# B&R Automation Studio project PloterCNC
Automation Studio 4.7.3.93 SP; technology packages: mapp 5.10.1, mappCockpit 5.10.1, mappControl 5.10.0, mappMotion 5.10.1, mappView 5.10.1

## Configuration PloterCNC

CPU X20CP3584, AutomationRuntime C4.72, Build 4.1.2, Safety 0.0, Vc V4.72.0

### Task classes (Cpu.sw)
```
Cyclic#2:
  Program <- Program.prg
DataObjects: McAcpSys
NcDataObjects: CncProg <- CncProg.dob, CncSquare <- CncSquare.dob
Binaries: udbdef, arsvcreg, FWRules, McAcpDrv, McMechSys, McAcpSim, mvLoader, mCoWebSc, TCData, arflatprv, arcoal, iomap, Config_4, asfw, Config_3, Role, Config_1, Config_2, arconfig, ashwd, Hierarchy, sysconf, User, ashwac
Libraries: McBase, MpCnc, MpBase, McAxGroup, McPathGen, McAxis, McProgInt, McAcpAx, CoTrace, AsZip, FileIO, runtime, asmem, sys_lib, arssl, asarprof, powerlnk, asieccon, dataobj, brsystem, asarlog, MpAlarmX, astime, MpServer
```

### Hardware
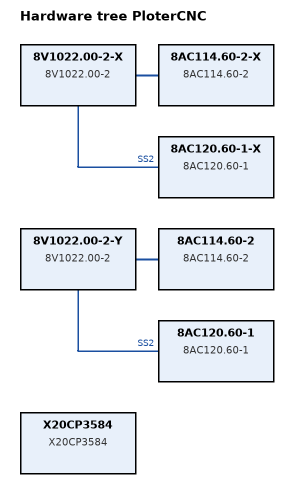
```
8AC114.60-2 : 8AC114.60-2 v1.0.0.8  [SS -> 8V1022.00-2-Y.SS1; PLK1 -> 8AC114.60-2-X.PLK2 [Cable Type=PowerlinkCable, Length=10, Version=1.0.0.2]]
8AC114.60-2-X : 8AC114.60-2 v1.0.0.8  [SS -> 8V1022.00-2-X.SS1; PLK1 -> X20CP3584.IF3 [Cable Type=PowerlinkCable, Length=10, Version=1.0.0.2]; PLK2 -> 8AC114.60-2.PLK1 [Cable Type=PowerlinkCable, Length=10, Version=1.0.0.2]]
8AC120.60-1 : 8AC120.60-1 v2.2.0.0  [SS -> 8V1022.00-2-Y.SS2]
  PlugInType = Encoder
  McAcoposTypeID = AcoposPlugInConfig
8AC120.60-1-X : 8AC120.60-1 v2.2.0.0  [SS -> 8V1022.00-2-X.SS2]
  PlugInType = Encoder
  McAcoposTypeID = AcoposPlugInConfig
8V1022.00-2-X : 8V1022.00-2 v2.2.0.0
  DriveConfiguration/Module:
    McAcoposTypeID = AcoposConfig
    ActivateACOPOSSimulationOnPLC = 0
  DriveConfiguration/Channel[1]/RealAxis:
    AxisReference = gAxisQX
  DriveConfiguration/Channel[1]/RealAxis/MechanicalElements/Gearbox:
    InputIsReadOnly = 0
    Input = 1
    OutputIsReadOnly = 0
    Output = 1
  DriveConfiguration/Channel[1]/RealAxis/MechanicalElements/RotaryToLinearTransformation:
    ReferenceDistanceIsReadOnly = 0
    ReferenceDistance = 1.385
  DriveConfiguration/Channel[1]/RealAxis/Controller:
    ModeIsReadOnly = 0
    Mode = PositionController
  DriveConfiguration/Channel[1]/RealAxis/Controller/Mode/Position:
    ProportionalGain = 454
    IntegrationTime = 0.0
    PredictionTime = 0.0004
    TotalDelayTime = 0.0004
  DriveConfiguration/Channel[1]/RealAxis/Controller/Mode/Speed:
    ProportionalGainIsReadOnly = 0
    ProportionalGain = 0.6499999
    IntegrationTimeIsReadOnly = 0
    IntegrationTime = 0.0
    FilterTimeIsReadOnly = 0
    FilterTime = 0.0
  DriveConfiguration/Channel[1]/RealAxis/Controller/Mode/LoopFilters:
    LoopFilter1 = NotUsed
    LoopFilter2 = NotUsed
    LoopFilter3 = NotUsed
  DriveConfiguration/Channel[1]/RealAxis/Homing:
    Mode = AbsoluteCorrection
  DriveConfiguration/Channel[1]/RealAxis/Homing/Mode:
    Position = -223
  DriveConfiguration/Channel[1]/RealAxis/Homing:
    RestorePositionVariable = 
  DriveConfiguration/Channel[1]/RealAxis/StopReaction:
    Quickstop = DecelerationLimit
    DriveError = DecelerationLimit
  DriveConfiguration/Channel[1]/RealAxis/MovementErrorLimits:
    PositionError = 1.0
    VelocityErrorMonitoring = Automatic1
  DriveConfiguration/Channel[1]/RealAxis:
    JerkFilter = NotUsed
  DriveConfiguration/Channel[1]/RealAxis/DigitalInputs/HomingSwitch:
    Level = High
  DriveConfiguration/Channel[1]/RealAxis/DigitalInputs/PositiveLimitSwitch:
    Level = Low
  DriveConfiguration/Channel[1]/RealAxis/DigitalInputs/NegativeLimitSwitch:
    Level = Low
  DriveConfiguration/Channel[1]/RealAxis/DigitalInputs/Trigger1:
    Level = High
  DriveConfiguration/Channel[1]/RealAxis/DigitalInputs/Trigger2:
    Level = High
  DriveConfiguration/Channel[1]/RealAxis/DigitalInputs/Quickstop:
    Input = Trigger2
  DriveConfiguration/Channel[1]/RealAxis/Simulation:
    SimulationModeOnPLC = SetValueGeneration
    SimulationModeOnACOPOS = NotUsed
8V1022.00-2-Y : 8V1022.00-2 v2.2.0.0
  DriveConfiguration/Module:
    McAcoposTypeID = AcoposConfig
    ActivateACOPOSSimulationOnPLC = 0
  DriveConfiguration/Channel[1]/RealAxis:
    AxisReference = gAxisQY
  DriveConfiguration/Channel[1]/RealAxis/MechanicalElements/Gearbox:
    InputIsReadOnly = 0
    Input = 1
    OutputIsReadOnly = 0
    Output = 1
  DriveConfiguration/Channel[1]/RealAxis/MechanicalElements/RotaryToLinearTransformation:
    ReferenceDistanceIsReadOnly = 0
    ReferenceDistance = 1.385
  DriveConfiguration/Channel[1]/RealAxis/Controller:
    ModeIsReadOnly = 0
    Mode = PositionController
  DriveConfiguration/Channel[1]/RealAxis/Controller/Mode/Position:
    ProportionalGain = 496
    IntegrationTime = 0.0
    PredictionTime = 0.0004
    TotalDelayTime = 0.0004
  DriveConfiguration/Channel[1]/RealAxis/Controller/Mode/Speed:
    ProportionalGainIsReadOnly = 0
    ProportionalGain = 0.8499999
    IntegrationTimeIsReadOnly = 0
    IntegrationTime = 0.0
    FilterTimeIsReadOnly = 0
    FilterTime = 0.0
  DriveConfiguration/Channel[1]/RealAxis/Controller/Mode/LoopFilters:
    LoopFilter1 = NotUsed
    LoopFilter2 = NotUsed
    LoopFilter3 = NotUsed
  DriveConfiguration/Channel[1]/RealAxis/Homing:
    Mode = AbsoluteCorrection
  DriveConfiguration/Channel[1]/RealAxis/Homing/Mode:
    Position = 1761
  DriveConfiguration/Channel[1]/RealAxis/Homing:
    RestorePositionVariable = 
  DriveConfiguration/Channel[1]/RealAxis/StopReaction:
    Quickstop = DecelerationLimit
    DriveError = DecelerationLimit
  DriveConfiguration/Channel[1]/RealAxis/MovementErrorLimits:
    PositionError = 1.0
    VelocityErrorMonitoring = Automatic1
  DriveConfiguration/Channel[1]/RealAxis:
    JerkFilter = NotUsed
  DriveConfiguration/Channel[1]/RealAxis/DigitalInputs/HomingSwitch:
    Level = High
  DriveConfiguration/Channel[1]/RealAxis/DigitalInputs/PositiveLimitSwitch:
    Level = Low
  DriveConfiguration/Channel[1]/RealAxis/DigitalInputs/NegativeLimitSwitch:
    Level = Low
  DriveConfiguration/Channel[1]/RealAxis/DigitalInputs/Trigger1:
    Level = High
  DriveConfiguration/Channel[1]/RealAxis/DigitalInputs/Trigger2:
    Level = High
  DriveConfiguration/Channel[1]/RealAxis/DigitalInputs/Quickstop:
    Input = Trigger2
  DriveConfiguration/Channel[1]/RealAxis/Simulation:
    SimulationModeOnPLC = SetValueGeneration
    SimulationModeOnACOPOS = NotUsed
X20CP3584 : X20CP3584 v1.6.0.0
  Connector IF2:
    ActivateDevice = 1
    Mode = Manual
    InternetAddress = 10.0.0.2
    SubnetMask = 255.255.255.0
  Connector IF3:
    Channel1
    ChannelID1 = McAcpBroadcast
    ChannelType1 = OCTET[96]
  ConfigurationID = PloterCNC_PloterCNC
  UserPartitionSize = 100
  Simulation = 1
  TimerDeviceType = EPLX2X
  TimerDevice = X20CP3584.IF3
  TaskClassIdleTime = 2000
  Cyclic1Duration = 2000
  Cyclic1Tolerance = 0
  FtpUser1
  FtpUsername1 = admin
  FtpUserPassword1 = uWZf7lfkDMUZL52pN0YGjFsSlLYs7TnNYj8rJpA5ubQ=  // admin
  FtpUserSalt1 = 89IIsKuO
  FTPAccessRight1 = 0
  ActivateOpcUa = 1
  OpcUaInformationModels_PV_Version = 1
```

### Config_1.axesgroup - X20CP3584/mappMotion/2AxesCNCXY/Config_1.axesgroup
```
Element gCncXY (Type=axesgroup)
  Type = PathGenAxesGroup
    ProcessingTaskClass = 1
    License = 1
    PhysicalAxes:
      JointAxes:
        JointAxis[1]:
          Name = QX
          AxisRef = gAxisQX
        JointAxis[2]:
          Name = QY
          AxisRef = gAxisQY
    MechanicalSystem:
      MechSysRef = MechSys_2AxCNCXY
    BasicSettings:
      ModalDataBehaviour = ResetToDefault
      GeometryPlanning:
        RoundingMode = Standard
        MaxCornerDeviation = 0.0
        MaxTangentialTransitionDeviation = 0.0
        MaxRadiusDeviation = 0.001
        WorkingPlane = XY
      TrajectoryPlanning = Basic
        LimitCheckResolution = UserDefinedTime
          Time = 0.01
        BufferTime = UserDefinedTime
          Time = 0.1
    AxesGroupFeatures:
      FeatureRef[1] = Feature_Programs
      FeatureRef[2] = Feature_Jogging
  Alarms = None
```

### Config_2.axis - X20CP3584/mappMotion/2AxesCNCXY/Config_2.axis
```
Element gAxisQX (Type=axis)
  BaseTypeIsReadOnly = 0
  BaseType = LinearBounded
    MeasurementUnit = 5066068
    MeasurementResolutionIsReadOnly = 0
    MeasurementResolution = 0.01
    CountDirectionIsReadOnly = 0
    CountDirection = Standard
  MovementLimitsIsReadOnly = 0
  MovementLimits = Internal
    Position:
      LowerLimitMin = -1.79769313486231E308
      UpperLimitMax = 1.79769313486231E308
      LowerLimit = -10
      UpperLimit = 540
    VelocityIsReadOnly = 0
    Velocity:
      VelocityMax = 3.4E38
      Velocity = 100
    AccelerationIsReadOnly = 0
    Acceleration:
      AccelerationMax = 3.4E38
      Acceleration = 1000
    DecelerationIsReadOnly = 0
    Deceleration:
      DecelerationMax = 3.4E38
      Deceleration = 1000
  Alarms = None
Element gAxisQY (Type=axis)
  BaseTypeIsReadOnly = 0
  BaseType = LinearBounded
    MeasurementUnit = 5066068
    MeasurementResolutionIsReadOnly = 0
    MeasurementResolution = 0.01
    CountDirectionIsReadOnly = 0
    CountDirection = Inverse
  MovementLimitsIsReadOnly = 0
  MovementLimits = Internal
    Position:
      LowerLimitMin = -1.79769313486231E308
      UpperLimitMax = 1.79769313486231E308
      LowerLimit = -10
      UpperLimit = 410
    VelocityIsReadOnly = 0
    Velocity:
      VelocityMax = 3.4E38
      Velocity = 100
    AccelerationIsReadOnly = 0
    Acceleration:
      AccelerationMax = 3.4E38
      Acceleration = 1000
    DecelerationIsReadOnly = 0
    Deceleration:
      DecelerationMax = 3.4E38
      Deceleration = 1000
  Alarms = None
```

### Config_3.mechanicalsystem - X20CP3584/mappMotion/2AxesCNCXY/Config_3.mechanicalsystem
```
Element MechSys_2AxCNCXY (Type=mechanicalsystem)
  Type = 2AxesCNC
    Subtype = 2AxesCNCXY
      CoordinatesNames = Default
        XCoordinateName = X
        YCoordinateName = Y
      WireFrameModel = Standard
        FlangeToTcp = ConnectionLine
          Distance = 0.0
      JointAxesPositionLimits:
        JointAxis[1] = UseAxisLimits
        JointAxis[2] = UseAxisLimits
```

### Config_4.axesgroupfeature - X20CP3584/mappMotion/2AxesCNCXY/Config_4.axesgroupfeature
```
Element Feature_Programs (Type=axesgroupfeature)
  Type = Program
    ModalDataBehaviour = UseAxesGroupSettings
    InitialSettings:
      InterpolationTypes = LinearRapid
      PositionCoordinates = Absolute
      CircleCoordinates = Relative
      JACS_ACSProgramming = JACS
      ContourConnection = Inactive
      ProgrammingUnits = UseAxesGroupSettings
      Feedrates:
        FeedCharacteristic = StandardCharacteristic
        FeedType = Feedrate
        FeedReduction = Inactive
        FeedrateValue = 0.0
        InverseFeedrateValue = 0.0
        FeedratePerRevValue = 0.0
    DefaultLanguage = BRGCode
    Location = Default
      FileDevice = CNC_PrgDir
Element Feature_Jogging (Type=axesgroupfeature)
  Type = Jogging
```

### Config.mpalarmxcore - X20CP3584/mappServices/Config.mpalarmxcore
```
Element gAlarmXCore (Type=mpalarmxcore)
  mapp.AlarmX.Core.Configuration:
    [0]:
      Name = XAxisOutOfBounds
      Message = X axis went out of bounds!
      Behavior = LevelMonitoring
        Monitoring:
          MonitoredPV = ::Program:MpCnc2Axis_0.X
          LowLimitEnable = Static
            Limit = 0
          HighLimitEnable = Static
            Limit = 540
    [1]:
      Name = UserAlarm
      Message = This alarm is set by user!
      Behavior = PersistentAlarm
```

## Logical view

Binary libraries used (declarations not repeated): operator, runtime, astime, AsIecCon, McBase, MpCnc 5.10.1, MpBase, McAxGroup 5.10.1, McPathGen 5.10.1, McAxis, McProgInt 5.10.1, McAcpAx, CoTrace, AsZip, FileIO, MpAlarmX 5.10.1, MpServer 5.10.0


### Data object Logical/CncProg (Cnc)

#### CncProg.cnc - CNC program (G-Code)
```
%001 (CncProgram)

N10 G90     (absolute coordinates)
N20 F3000    (Feed rate in measurements units/min)

N30 G04 2   (dwell time 2s)

N50 G01 X80 Y100  (linear move)

N60 G04 2         (dwell time 2s)

N100 G00 X0 Y0    (rapid move to zero)
N999 M30
```

### Program Logical/Program (IEC)

#### Types.typ
```iecst
TYPE
	MotionStep_type :
		(
		STEP_INIT,
		STEP_POWER,
		STEP_HOME,
		STEP_AWAIT,
		STEP_RUN_PROGRAM,
		STEP_PROGRAM_INTERRUPTED,
		STEP_MOVE_Y_AXIS,
		STEP_MOVE_X_AXIS,
		STEP_ERROR
		);
END_TYPE
```

#### Variables.var
```iecst
VAR
	MpAlarmXHistory_0 : MpAlarmXHistory;
	MpAlarmXCore_0 : MpAlarmXCore;
	MpCnc2Axis_0 : MpCnc2Axis;
	CncParameters : MpCnc2AxisParType;
	MotionStep : MotionStep_type;
	ProgramOption : BOOL;
	AxisVelocity : REAL := 0.0;
END_VAR
(*Comands*)
VAR
	diErrorReset : BOOL;
	diRunProgram : BOOL;
	diResumeProgram : BOOL;
	diInterruptProgram : BOOL;
	diIncreaseYAxis : BOOL;
	diDecreaseYAxis : BOOL;
	diIncreaseXAxis : BOOL;
	diDecreaseXAxis : BOOL;
	diStop : BOOL;
	diStart : BOOL;
END_VAR
```

#### Main.st
```iecst
PROGRAM _INIT
	MpAlarmXCore_0.MpLink := ADR(gAlarmXCore);
	MpAlarmXCore_0.Enable := TRUE;

	MpAlarmXHistory_0.MpLink := ADR(gAlarmXHistory);
	MpAlarmXHistory_0.Enable := TRUE;

	MpCnc2Axis_0.MpLink := ADR(gCncXY);
	MpCnc2Axis_0.Enable := TRUE;
	MpCnc2Axis_0.Parameters := ADR(CncParameters);

	MpCnc2Axis_0.Override := 100.0;
	AxisVelocity := 0;
	CncParameters.Jog.Velocity[0] := AxisVelocity;
	CncParameters.Jog.Velocity[1] := AxisVelocity;
END_PROGRAM

PROGRAM _CYCLIC

	IF ProgramOption THEN
		CncParameters.ProgramName := 'CncSquare';
	ELSE
		CncParameters.ProgramName := 'CncProg';
	END_IF;

	MpCnc2Axis_0.ErrorReset := diErrorReset;

	IF EDGEPOS(MpCnc2Axis_0.Error) THEN
		MotionStep := STEP_ERROR;
	END_IF;

	CASE MotionStep OF
		STEP_INIT:
			MpCnc2Axis_0.Power := FALSE;
			MpCnc2Axis_0.Home := FALSE;

			IF diStart THEN
				MotionStep := STEP_POWER;
			END_IF;
		STEP_POWER:
			MpCnc2Axis_0.Power := TRUE;

			IF MpCnc2Axis_0.PowerOn THEN
				MotionStep := STEP_HOME;
			END_IF;
		STEP_HOME:
			MpCnc2Axis_0.Home := TRUE;

			IF MpCnc2Axis_0.IsHomed THEN
				MotionStep := STEP_AWAIT;
			END_IF;
		STEP_AWAIT:

			IF diStop THEN
	  			MotionStep := STEP_INIT;
			ELSIF diRunProgram THEN
				MotionStep := STEP_RUN_PROGRAM;
			ELSIF diIncreaseXAxis THEN
				CncParameters.Jog.Velocity[0] := AxisVelocity;
				MotionStep := STEP_MOVE_X_AXIS;
			ELSIF diDecreaseXAxis THEN
				CncParameters.Jog.Velocity[0] := -AxisVelocity;
				MotionStep := STEP_MOVE_X_AXIS;
			ELSIF diIncreaseYAxis THEN
				CncParameters.Jog.Velocity[1] := AxisVelocity;
				MotionStep := STEP_MOVE_Y_AXIS;
			ELSIF diDecreaseYAxis THEN
				CncParameters.Jog.Velocity[1] := -AxisVelocity;
				MotionStep := STEP_MOVE_Y_AXIS;
			END_IF;
		STEP_RUN_PROGRAM:
			MpCnc2Axis_0.MoveProgram := TRUE;
			MpCnc2Axis_0.Continue := FALSE;

			IF MpCnc2Axis_0.MoveDone THEN
				MotionStep := STEP_AWAIT;
				MpCnc2Axis_0.MoveProgram := FALSE;
			END_IF;

			IF diInterruptProgram THEN
				MotionStep := STEP_PROGRAM_INTERRUPTED;
			END_IF;
		STEP_PROGRAM_INTERRUPTED:
			MpCnc2Axis_0.Interrupt := TRUE;

			IF diResumeProgram THEN
				MotionStep := STEP_RUN_PROGRAM;
				MpCnc2Axis_0.Interrupt := FALSE;
				MpCnc2Axis_0.Continue := TRUE;
			END_IF;
		STEP_MOVE_X_AXIS:
			MpCnc2Axis_0.Jog := TRUE;

			IF NOT(diIncreaseXAxis) AND NOT(diDecreaseXAxis) THEN
				MotionStep := STEP_AWAIT;
				MpCnc2Axis_0.Jog := FALSE;
				CncParameters.Jog.Velocity[0] := 0;
			END_IF;
		STEP_MOVE_Y_AXIS:
			MpCnc2Axis_0.Jog := TRUE;

			IF  NOT(diIncreaseYAxis) AND NOT(diDecreaseYAxis) THEN
				MotionStep := STEP_AWAIT;
				MpCnc2Axis_0.Jog := FALSE;
				CncParameters.Jog.Velocity[1] := 0;
			END_IF;
		STEP_ERROR:

			IF NOT(MpCnc2Axis_0.Error) THEN
	  			MotionStep := STEP_INIT;
			END_IF;
	END_CASE;

	MpAlarmXHistory_0();
	MpAlarmXCore_0();
	MpCnc2Axis_0();
END_PROGRAM

PROGRAM _EXIT

	MpCnc2Axis_0.Power  := FALSE;
	MpCnc2Axis_0.Home   := FALSE;
	MpCnc2Axis_0();

	MpCnc2Axis_0.Enable := FALSE;
	MpCnc2Axis_0();

END_PROGRAM
```

### Data object Logical/CncSquare (Cnc)

#### CncSquare.cnc - CNC program (G-Code)
```
%001 (CncSquare)

N10 G91     (absolute coordinates)
N20 F1200    (Feed rate in measurements units/min)

N30 G04 2   (dwell time 2s)

N50 G01 X0 Y100  (linear move)

N60 G04 1

N70 G01 X100 Y0  (linear move)

N80 G04 1         (

N90 G01 X0 Y-100  (linear move)

N100 G04 1

N110 G01 X-100 Y0  (linear move)

N200 G00 X0 Y0    (rapid move to zero)
N999 M30
```

- Visualisation Logical/mappView (not shown)

Listed in the project but not available here: Logical/Global.typ, Logical/Global.var
